// TIA Portal V20 export
DATA_BLOCK "HmiInterface"   // DB145
// stored: Access Published, MemoryReserve 100, Namespace Unit1.Em11
   VAR
      em : "LAF_typeEmInterface";
      weightCheck : "LER_typeSequenceInterface";
      cmWeightCheckJRDetect : "LBC_typeDigitalSignalInterface";
      cmWeightCheckControl : "LER_WeightCheckInterface";
   END_VAR
   VAR RETAIN
      cmWeightCheckHistory : "LER_typeWeightCheckHistory";
   END_VAR
   VAR
      "=====미사용=====" { ExternalAccessible := 'False'; ExternalVisible := 'False'; ExternalWritable := 'False'} : Bool;
      cmWeightCheckStageLiftUpDown : "LBC_typeTwoWayActuatorInterface";
   END_VAR
BEGIN
   cmWeightCheckControl.configuration.hwID.pncMainControlID := 612;
   cmWeightCheckControl.configuration.hwID.pncMainStatusID := 612;
   cmWeightCheckControl.configuration.hwID.scaleControlID := 613;
   cmWeightCheckControl.configuration.hwID.scaleStatusID := 613;
END_DATA_BLOCK
